// TIA Portal V20 export
DATA_BLOCK "PNDevDiagStatus"   // DB96
// stored: InstanceOfName LER_DiagnosticsInterface, InstanceOfType UDT
"LER_DiagnosticsInterface"
   // VAR
   //    DevState { S7_SetPoint := 'True'} : "LER_DevState";
   //    DigState { S7_SetPoint := 'True'} : Array[0..15] of Bool;
   //    Station_Position : Int;
   // END_VAR
BEGIN
END_DATA_BLOCK
